// TIA Portal V20 export
FUNCTION_BLOCK "SysPnSlaveDeactivate"   // FB2500, FBD
TITLE = Profinet Slave Deactivate / manage a sensor
{ S7_Optimized_Access := 'TRUE' }
AUTHOR : MiCROTEC
VERSION : 1.5
// -2018.12 : Martin
// stored: AutoNumber false, MemoryReserve 100, SetENOAutomatically false
   VAR_INPUT
      iSlave { ExternalAccessible := 'False'; ExternalVisible := 'False'; ExternalWritable := 'False'} : HW_DEVICE;
      iDeactivate { ExternalAccessible := 'False'; ExternalVisible := 'False'; ExternalWritable := 'False'} : Bool;
   END_VAR
   VAR_OUTPUT
      oSlaveActive { ExternalAccessible := 'False'; ExternalVisible := 'False'; ExternalWritable := 'False'} : Bool;   // Sensor fault , sensor is broken or is dirty
      oError { ExternalAccessible := 'False'; ExternalVisible := 'False'; ExternalWritable := 'False'} : Bool;   // Sensor fault , was to long occupied, maybe dirty or misaligned
   END_VAR
   VAR
      var { ExternalAccessible := 'False'; ExternalVisible := 'False'; ExternalWritable := 'False'} : Struct
         "bool" : Bool;
         "byte" : Byte;
         "word" : Word;
         "dword" : DWord;
         "int" : Int;
         "dint" : DInt;
         "real" : Real;
         s5time : S5Time;
         "time" : Time;
         hm : Array[1..16] of Bool;
         fm : Array[1..16] of Bool;
      END_STRUCT;
      vInit { ExternalAccessible := 'False'; ExternalVisible := 'False'; ExternalWritable := 'False'} : Bool;
      vStart { ExternalAccessible := 'False'; ExternalVisible := 'False'; ExternalWritable := 'False'} : Bool;
      vBusy { ExternalAccessible := 'False'; ExternalVisible := 'False'; ExternalWritable := 'False'} : Bool;
      vMode { ExternalAccessible := 'False'; ExternalVisible := 'False'; ExternalWritable := 'False'} : USInt;   // // 0: Status 1: aktivieren 2: deaktivieren
      vStep { ExternalAccessible := 'False'; ExternalVisible := 'False'; ExternalWritable := 'False'} : Int;
      vRetval { ExternalAccessible := 'False'; ExternalVisible := 'False'; ExternalWritable := 'False'} : Word;
   END_VAR
BEGIN

REGION Network 1 (SCL)
   CASE #vStep OF
       0:(*Init*)
           IF NOT #vInit OR #oError THEN
               #vStep := 110;
           ELSIF #oSlaveActive <> NOT #iDeactivate THEN
               #vStep := 10;
           END_IF;

       10:(*Aktiviere/Deaktiviere Slave*)
           #vStart := true;
           IF #iDeactivate THEN
               #vMode := 2;
           ELSE
               #vMode := 1;
           END_IF;
           #vStep := 20;

       20:(*Warte bis Fertig*)
           IF NOT #vBusy THEN
               #vStep := 30;
           END_IF;

       30:(*fertig*)
           #oError := #vRetval >= W#16#8000;
           #vStart := FALSE;
           #vStep := 110;

       110: (*Status holen*)
           #vStart := true;
           #vMode := 0;
           #vStep := 120;

       120:(*Warte bis Fertig*)
           IF NOT #vBusy THEN
               #vStep := 130;
           END_IF;

       130:(*fertig*)
           #oSlaveActive := #vRetval = 1;
           #oError := #vRetval >= W#16#8000;
           #vStart := FALSE;
           #vInit := true;
           #vStep := 0;


   END_CASE;

   #vRetval := D_ACT_DP(REQ := #vStart, MODE := #vMode, LADDR := #iSlave, BUSY => #vBusy);
END_REGION
END_FUNCTION_BLOCK
